FUNCTION_BLOCK Agent_1 (* JADE Implementation *)
  (* Standard: 61499-1 *)
  (* Version 1.0, 2015-04-13, Sadik, FraunhoferIGD *)
  (* Compiler header: package fb.rt; *)
  (* Compiler Java Sun JDK 1.5.0 *)
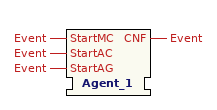
  EVENT_INPUT
    StartMC; (* Normal Execution Request *)
    StartAC; (* Normal Execution Request *)
    StartAG; (* Normal Execution Request *)
  END_EVENT
  EVENT_OUTPUT
    CNF; (* Execution Confirmation *)
  END_EVENT
END_FUNCTION_BLOCK
